PROGRAM state_transition
VAR PERSISTENT
	//Hard coded state values for comparison
	state_faulted : INT :=0;
	state_stopped : INT :=10;
	state_idle : INT :=20;
	state_cip : INT :=30;
	state_manual : INT :=40;
	state_maint : INT :=50;
	state_active_input : INT :=61;
	state_active_conc : INT :=62;
	state_active_opt : INT :=63;
	
END_VAR

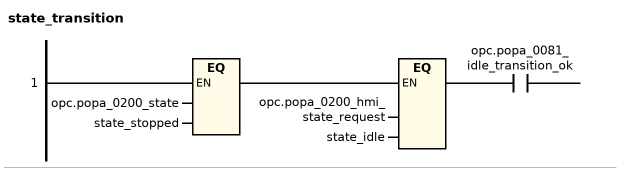
// NETWORK 1
(* (opc.popa_0200_state = state_stopped AND opc.popa_0200_hmi_state_request = state_idle) AND opc.popa_0081_idle_transition_ok; result not used *)

END_PROGRAM

(* stored: Version 1.1.0.1, ProductVersion 3.1.4024.12
   POU state_transition: Id {48687b9f-7057-49bd-b80e-9cc206fe590e}, SpecialFunc None *)
